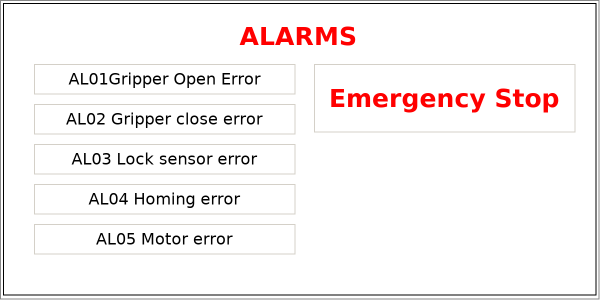
VISUALIZATION Alarm  // 600x300
    Rectangle (3,3 593x292)
    Label (217,21 163x30), "ALARMS"
    Textfield (34,64 261x30), "AL01Gripper Open Error", invisible if: GVL_IO.Gripper_Open_Error = 0
    Textfield (34,104 261x30), "AL02 Gripper close error", invisible if: GVL_IO.Gripper_Close_Error = 0
    Textfield (34,144 261x30), "AL03 Lock sensor error", invisible if: GVL_IO.SensorLock_Error = 0
    Textfield (34,184 261x30), "AL04 Homing error", invisible if: GVL_IO.Homing_Error = 0
    Textfield (34,224 261x30), "AL05 Motor error", invisible if: GVL_IO.Motor_Error = 0
    Textfield (314,64 261x68), "Emergency Stop", invisible if: GVL_IO.ixEmergancy_Stop
END_VISUALIZATION

(* stored: Version 1.1.0.1, ProductVersion 3.1.4024.13
   Visu Alarm: Id {ab34ea3a-99e0-4caa-81ba-d98874a3afec} *)
